// TIA Portal V21 export
TYPE "coneCrusherConfigs"
   STRUCT
      self : "coneCrusherConfig";
      luS : "lubricationSystemConfigs";
      sg : "switchgearConfig";
      btnStart : "LBC_typeDigitalSignalConfiguration";
      btnStop : "LBC_typeDigitalSignalConfiguration";
      keySwitch : "LBC_typeDigitalSignalConfiguration";
      emStop : "LBC_typeDigitalSignalConfiguration";
      btnReset : "LBC_typeDigitalSignalConfiguration";
      btnStartLuS : "LBC_typeDigitalSignalConfiguration";
      btnStopLuS : "LBC_typeDigitalSignalConfiguration";
      premoldingSw : "LBC_typeDigitalSignalConfiguration";
      crusherEccentricTemp : "LBC_typeAnalogInputConfiguration";
      crusherOuterBearingTemp : "LBC_typeAnalogInputConfiguration";
      crusherInnerBearingTemp : "LBC_typeAnalogInputConfiguration";
      driveFrontBearingTemp : "LBC_typeAnalogInputConfiguration";
      driveRearBearingTemp : "LBC_typeAnalogInputConfiguration";
      driveWindingTempP1 : "LBC_typeAnalogInputConfiguration";
      driveWindingTempP2 : "LBC_typeAnalogInputConfiguration";
      driveWindingTempP3 : "LBC_typeAnalogInputConfiguration";
      driveCurrent : "LBC_typeAnalogInputConfiguration";
      sgReady { S7_SetPoint := 'True'} : "LBC_typeDigitalSignalConfiguration";
      sgFbOn { S7_SetPoint := 'True'} : "LBC_typeDigitalSignalConfiguration";
      sgFbOff { S7_SetPoint := 'True'} : "LBC_typeDigitalSignalConfiguration";
      sgStart : "LBC_typeDigitalSignalConfiguration";
      sgStop : "LBC_typeDigitalSignalConfiguration";
      preStartAlmOn : "LBC_typeDigitalSignalConfiguration";
      feedEn : "LBC_typeDigitalSignalConfiguration";   // Allow feed from upstream unit
      preStartAlmFb { S7_SetPoint := 'True'} : "LBC_typeDigitalSignalConfiguration";
   END_STRUCT;
END_TYPE
